// TIA Portal V20 export
ORGANIZATION_BLOCK "Main"   // OB1001, LAD, ProgramCycle
TITLE = "Main Program Sweep (Cycle)"
AUTHOR : ERsystem_FA2_DH. Kim
// stored: AutoNumber false, IsIECCheckEnabled true, Namespace Unit1, SetENOAutomatically false
   VAR_INPUT
      Initial_Call : Bool;   // Initial call of this OB
      Remanence : Bool;   // =True, if remanent data are available
   END_VAR
   VAR_TEMP
      tempIndex : Int;   // Index of Unit in the array
   END_VAR
BEGIN

REGION Network 1: Call Unit
   // Assign the number of the unit to a temp for correct array index access.
   // Number is defined in PLC tags of Software Unit Global.
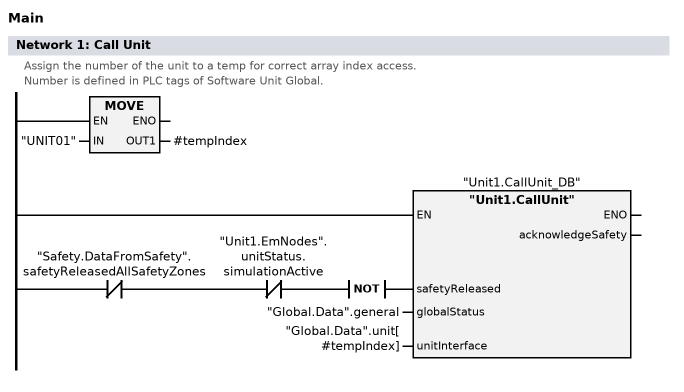
   RUNG wire#powerrail
      Move(in := "UNIT01", out1 => #tempIndex)
   END_RUNG
   RUNG wire#powerrail
      "Unit1.CallUnit_DB"(safetyReleased := wire#w1, globalStatus := "Global.Data".general, unitInterface := "Global.Data".unit[#tempIndex], acknowledgeSafety =>)
   END_RUNG
   RUNG wire#powerrail
      I_Contact( "Safety.DataFromSafety".safetyReleasedAllSafetyZones )
      I_Contact( "Unit1.EmNodes".unitStatus.simulationActive )
      Not()
   END_RUNG wire#w1
   // the same network as SCL:
   #tempIndex := "UNIT01";
   "Unit1.CallUnit_DB"(safetyReleased := NOT (NOT "Safety.DataFromSafety".safetyReleasedAllSafetyZones AND NOT "Unit1.EmNodes".unitStatus.simulationActive),   // "Unit1.CallUnit"
                       globalStatus := "Global.Data".general,
                       unitInterface := "Global.Data".unit[#tempIndex]);
END_REGION
END_ORGANIZATION_BLOCK
